// TIA Portal V20 export
VAR_GLOBAL   // PLC tag table "PLC_Centralizer_PLC_Production_And_Rework"
   In_PLC_Production_And_Rework AT %I500.0 : "IO_Device_Conveyor_Belt_Input";
   Out_PLC_Production_And_Rework AT %Q500.0 : "IO_Device_Conveyor_Belt_Ouput";
END_VAR
